// TIA Portal V19 export
VAR_GLOBAL   // PLC tag table "Equipment_Template_DefaultTagTable_2"
   "Tag_49(4)" AT %I30042.0 : Bool;   // 物流线允许出
   "Tag_50(4)" AT %I30042.1 : Bool;   // 物流线通知托盘送出完成
   "Tag_51(4)" AT %I30042.2 : Bool;   // 物流线收到单机收到的物流线出到位信号
   "Tag_52(4)" AT %I30042.3 : Bool;   // 物流线空闲
   "Tag_53(4)" AT %I30042.4 : Bool;
   "Tag_54(4)" AT %I30042.5 : Bool;
   "Tag_55(4)" AT %I30042.6 : Bool;
   "Tag_56(4)" AT %I30042.7 : Bool;   // 物流请求出托盘
   "Tag_57(4)" AT %I30043.0 : Bool;   // 物流线忙碌
   "Tag_58(4)" AT %I30043.1 : Bool;   // 物流线收到单机返回出到位信号
   "Tag_59(4)" AT %I30043.2 : Bool;   // 物流工位报警
   "Tag_60(4)" AT %I30043.3 : Bool;   // 物流有拖盘待出
   "Tag_61(4)" AT %I30043.4 : Bool;
   "Tag_62(4)" AT %I30043.5 : Bool;
   "Tag_63(4)" AT %I30043.6 : Bool;
   "Tag_64(4)" AT %I30043.7 : Bool;
   Tag_1 AT %M10000.0 : Bool;
END_VAR
